(* PLC project PLC, Beckhoff Automation GmbH TwinCAT PLC Control 3.5.13.21 *)
(* stored: creationDateTime 2024-02-17T22:43:21.1008995, modificationDateTime 2024-02-17T22:43:21.1008995 *)

TYPE PBStatus :
STRUCT
	name: STRING(G.nameStringLength);
	pushed: BOOL;
END_STRUCT
END_TYPE
